{attribute 'qualified_only'}
{attribute 'strict'}
TYPE RESET_STATE :
(
	IDLE,
	ERRACK_ON,
	ERRACK_OFF,
	IDLE2,
	ESTOP_RESET_ON
);
END_TYPE

(* stored: Version 1.1.0.1, ProductVersion 3.1.4022.12
   DUT RESET_STATE: Id {1d584288-8313-4925-b5af-cea35283fb22} *)
